// TIA Portal project "Project1" (V16)

(* hardware
DEVICE "S7-1200 station_1"  S7-1200 Station
   slot 0: "Rack_0"  S7-1200 Rack  Rack  V1.0
   slot 1: "PLC_1"  CPU 1214C AC/DC/Rly  6ES7 214-1BG40-0XB0  V4.2
*)

// ===== PLC "PLC_1"  CPU 1214C AC/DC/Rly =====

VAR_GLOBAL   // PLC tag table "Default tag table"
   ""Stop"" AT %I1.2 : Bool;
   ""Start"" AT %I1.1 : Bool;
   ""Tag_5"" AT %I0.1 : Bool;
   ""Quay_thuan"" AT %Q0.6 : Bool;
   ""Quay_nguoc"" AT %Q0.7 : Bool;
   ""Tag_3"" AT %Q8.1 : Bool;
END_VAR